PROGRAM pouS5Prompts
VAR
	


idbMsgPrompt: FB_CheckMessageBounds;
END_VAR

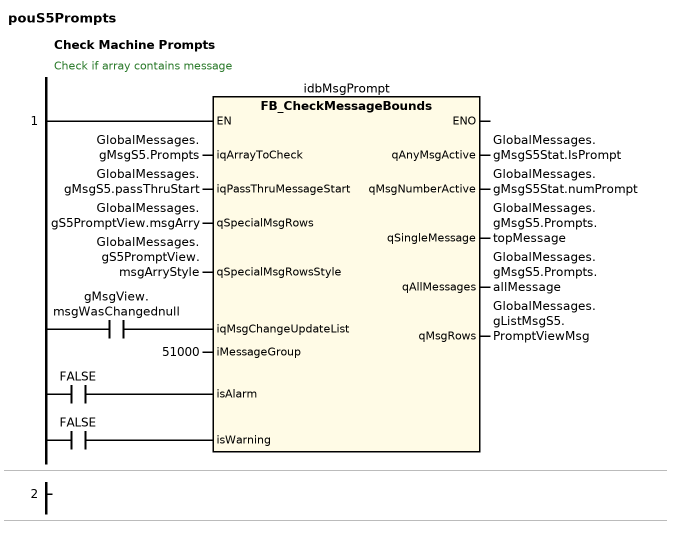
// NETWORK 1: Check Machine Prompts
// Check if array contains message
idbMsgPrompt(
    iqArrayToCheck := GlobalMessages.gMsgS5.Prompts,
    iqPassThruMessageStart := GlobalMessages.gMsgS5.passThruStart,
    qSpecialMsgRows := GlobalMessages.gS5PromptView.msgArry,
    qSpecialMsgRowsStyle := GlobalMessages.gS5PromptView.msgArryStyle,
    iqMsgChangeUpdateList := gMsgView.msgWasChangednull,
    iMessageGroup := 51000,
    isAlarm := FALSE,
    isWarning := FALSE,
    qAnyMsgActive => GlobalMessages.gMsgS5Stat.IsPrompt,
    qMsgNumberActive => GlobalMessages.gMsgS5Stat.numPrompt,
    qSingleMessage => GlobalMessages.gMsgS5.Prompts.topMessage,
    qAllMessages => GlobalMessages.gMsgS5.Prompts.allMessage,
    qMsgRows => GlobalMessages.gListMsgS5.PromptViewMsg); // FB_CheckMessageBounds

// NETWORK 2

END_PROGRAM

(* stored: Version 1.1.0.1, ProductVersion 3.1.4024.11
   POU pouS5Prompts: Id {bc0bd697-4d36-44ee-a168-cb9bd83cbb84}, SpecialFunc None *)
